{attribute 'GeneratedUsingTerminal: AT2050-0500-0020'}
{attribute addProperty BoxType "AT2050-0500-0020"}
{attribute addProperty Id "A_0093_AT2020_5250_0019_AT2020_5250AT2020_33A3DF1B80"}
{attribute addProperty CRC "2605914958"}
{attribute addProperty Size "80"}
TYPE A_0051_AT2050_0500_0020_9B531B4E EXTENDS AT2050_A7FEA1CF :
STRUCT
	{attribute addProperty Name "A_0093_AT2020_5250_0019_AT2020_5250"}
	{attribute addProperty PreviousPort "A_0051(AT2050-0500-0020) : B"}
	A_0093_AT2020_5250_0019_AT2020_5250 : AT2020_33A3DF1B;
END_STRUCT
END_TYPE

(* stored: Version 1.2.0.0, ProductVersion 3.1.4024.9
   DUT A_0051_AT2050_0500_0020_9B531B4E: Id {6dc45233-ba4e-4d6f-a09d-9cf98d80618b} *)
